FUNCTION_BLOCK FB_HeavyWash IMPLEMENTS I_WashStrategy

METHOD GetDuration : TIME
GetDuration := T#15S;
END_METHOD

METHOD Start 
VAR_IN_OUT
    config : ST_MachineConfig;
END_VAR
config.iDrumSpeed := 1200;
config.iWaterTemperature := 45;
END_METHOD

END_FUNCTION_BLOCK

(* stored: Version 1.1.0.1, ProductVersion 3.1.4024.16
   POU FB_HeavyWash: Id {e41f415f-ba68-4a16-b24e-7938e1f421e0}, SpecialFunc None
   Method GetDuration: Id {4231f7a7-eb2e-4f9b-a03f-aff44c0b572d}
   Method Start: Id {4bd65df7-22f1-4509-9f4d-5e228f44e99b} *)
